FUNCTION_BLOCK DeviceTypeDecode (* Basic Function Block Type *)
  (* Standard: 61499-2 *)
  (* Version 0.0, 6/4/2026, Schneider Electric, Template *)
  PACKAGE SE.Nereda;
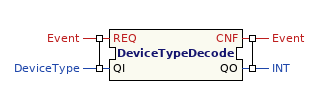
  EVENT_INPUT
    REQ WITH QI; (* Normal Execution Request *)
  END_EVENT
  EVENT_OUTPUT
    CNF WITH QO; (* Execution Confirmation *)
  END_EVENT
  VAR_INPUT
    QI : DeviceType; (* Input event qualifier *)
  END_VAR
  VAR_OUTPUT
    QO : INT; (* =1 : Motor ; =2 : Valve *)
  END_VAR
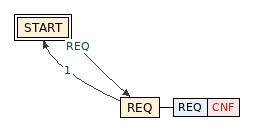
  EC_STATES
    START; (* Initial State *)
    REQ : REQ -> CNF; (* Normal execution *)
  END_STATES
  EC_TRANSITIONS
    START TO REQ := REQ;
    REQ TO START := 1;
  END_TRANSITIONS
  ALGORITHM REQ IN ST: (* Normally executed algorithm *)
;
IF QI = DeviceType#Motor THEN
	QO := 1;
ELSIF QI = DeviceType#Valve THEN
	QO := 2;
END_IF;
  END_ALGORITHM
END_FUNCTION_BLOCK
